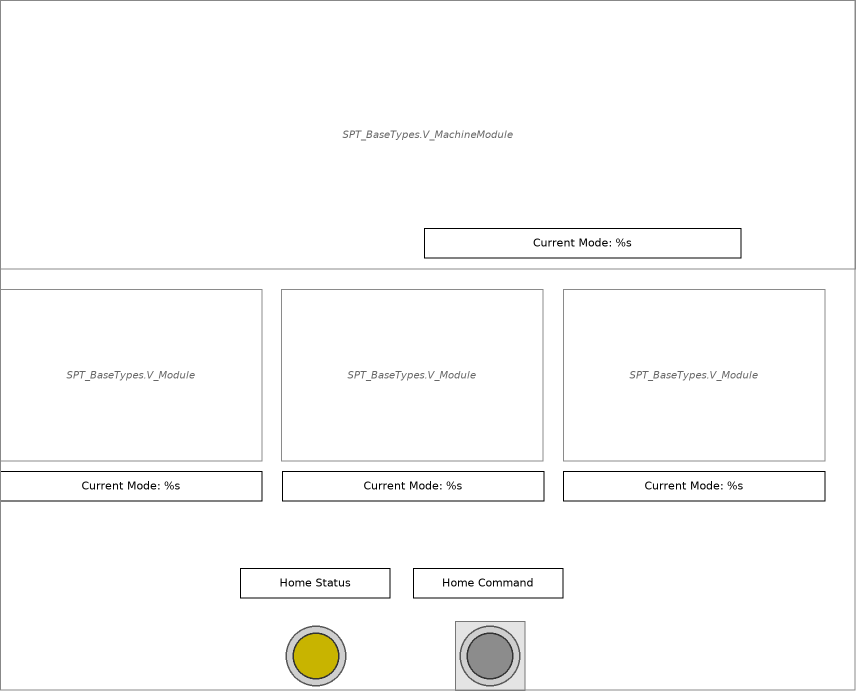
VISUALIZATION Visualization  // 856x691
    Frame (0,0 856x269)
        shows SPT_BaseTypes.V_MachineModule(HMI := MAIN.Machine.PackMLBaseModule_HMI)
    Lamp1 (281,621 70x70), variable: MAIN.Machine.Machine_HMI.Status.HomeComplete, style: Lamp-Lamp1-Yellow
    PushSwitch (455,621 70x70), variable: MAIN.Machine.Machine_HMI.Command.StartHoming, behaviour: TOGGLE, style: Switch-PushSwitch-Gray
    Rectangle (240,568 150x30), "Home Status"
    Rectangle (413,568 150x30), "Home Command"
    Frame (0,289 262x172)
        shows SPT_BaseTypes.V_Module(HMI := MAIN.Machine.Infeed.PackMLBaseModule_HMI)
    Frame (281,289 262x172)
        shows SPT_BaseTypes.V_Module(HMI := MAIN.Machine.Process.PackMLBaseModule_HMI)
    Frame (563,289 262x172)
        shows SPT_BaseTypes.V_Module(HMI := MAIN.Machine.Outfeed.PackMLBaseModule_HMI)
    Rectangle (424,228 317x30), "Current Mode: %s", text variable: MAIN.Machine.CurrentCustomMode
    Rectangle (0,471 262x30), "Current Mode: %s", text variable: MAIN.Machine.Infeed.CurrentCustomMode
    Rectangle (282,471 262x30), "Current Mode: %s", text variable: MAIN.Machine.Process.CurrentCustomMode
    Rectangle (563,471 262x30), "Current Mode: %s", text variable: MAIN.Machine.Outfeed.CurrentCustomMode
END_VISUALIZATION

(* stored: Version 1.1.0.1
   Visu Visualization: Id {e95e899b-b348-4b8e-9b57-7cb99c02523f} *)
